{attribute 'qualified_only'}
{attribute 'to_string'}
TYPE E_GCSpinAxisMoveAbsErrorCode :
(
	None := 0,
	Axis_Not_Servo_On_During_Starting,
	Axis_Is_Busy_During_Starting,
	Invalid_Param,
	MoveAbs_Error_During_Execute,
	Error_While_Stop_Axis
)UDINT;
END_TYPE

(* stored: Version 1.1.0.1, ProductVersion 3.1.4026.18
   DUT E_GCSpinAxisMoveAbsErrorCode: Id {8059fae9-a974-463c-9b89-43dd41b2bcf8} *)
